// TIA Portal project "010-sps_KnightRider_LightSequencer_tia-portal" (V17)

(* hardware
DEVICE "S7-300/ET200M-Station_1"  S7-300 station
   slot 0: "Profilschiene_0"  Rail  6ES7 390-1***0-0AA0
   slot 1: "PS 307 5A_1"  PS 307 5A  6ES7 307-1EA01-0AA0
   slot 2: "PLC_1"  CPU 314C-2 DP  6ES7 314-6CH04-0AB0  V3.3
      slot 0: "MPI-Schnittstelle_1"  MPI
      slot 1: "DP-Schnittstelle_1"  DP
      slot 2: "DI 24/DO 16_1"  DI24/DO16
      slot 3: "AI 5/AO 2_1"  AI5/AO2
      slot 4: "Zählen_1"  Counter
      slot 5: "Positionieren_1"  Positioning
   slot 4: "DI 16/DO 16x24VDC/0.5A_1"  DI16/DO16 x 24V / 0.5A  6ES7 323-1BL00-0AA0
   slot 5: "DI 16x24VDC_1"  DI16 x 24VDC  6ES7 321-1BH02-0AA0
   slot 6: "CP 342-5_1"  CP 342-5  6GK7 342-5DA03-0XE0  V6.0
   slot 7: "CP 343-1_1"  CP 343-1  6GK7 343-1EX30-0XE0  V2.0
*)

// ===== PLC "PLC_1"  CPU 314C-2 DP =====

VAR_GLOBAL   // PLC tag table "Standard-Variablentabelle"
   "Tag_3" AT %M255.1 : Bool;
   "Start" AT %E0.0 : Bool;
   "Tag_4" AT %M0.0 : Bool;
   "Tag_5" AT %MD10 : DWord;
   "Tag_6" AT %M20.0 : Bool;
   "Tag_7" AT %M0.1 : Bool;
   "Tag_8" AT %M0.2 : Bool;
   "Tag_1" AT %MD30 : DWord;
   "Ausgang" AT %AW0 : Word;
   "Tag_2" AT %AW2 : Word;
   "Tag_9" AT %M255.5 : Bool;
   "Tag_10" AT %M255.3 : Bool;
   "Tag_11" AT %A0.0 : Bool;
   "Tag_12" AT %A124.0 : Bool;
   "Tag_13" AT %A125.0 : Bool;
   "Tag_14" AT %A0.1 : Bool;
END_VAR

DATA_BLOCK "idb10 – Rotieren nach rechts"   // DB10
{ S7_Optimized_Access := 'FALSE' }
VERSION : 0.1
// stored: InstanceOfName FB10 – Rotieren nach rechts-links
"FB10 – Rotieren nach rechts-links"
BEGIN
END_DATA_BLOCK

DATA_BLOCK "idb13 – Lauflichtsteuerung"   // DB13
{ S7_Optimized_Access := 'FALSE' }
VERSION : 0.1
// stored: InstanceOfName FB13 – Lauflichtsteuerung
"FB13 – Lauflichtsteuerung"
BEGIN
END_DATA_BLOCK

DATA_BLOCK "idb15 Night Rider"   // DB15
{ S7_Optimized_Access := 'FALSE' }
VERSION : 0.1
// stored: InstanceOfName FB15 Night Rider
"FB15 Night Rider"
BEGIN
END_DATA_BLOCK

DATA_BLOCK "xdb100 VAR"   // DB100
{ S7_Optimized_Access := 'FALSE' }
VERSION : 0.1
   VAR
      x_Start : Bool;
      w_Src : Word := 1;
      x_clock : Bool;
      w_dest : Word;
   END_VAR
BEGIN
END_DATA_BLOCK

FUNCTION_BLOCK "FB10 – Rotieren nach rechts-links"   // FB10, FBD
{ S7_Optimized_Access := 'FALSE' }
VERSION : 0.1
   VAR_INPUT
      "xStep Val" : Int := 1;
      xClock : Bool;
      xRotierenRechts : Bool;
   END_VAR
   VAR_IN_OUT
      "dw Out Val" : DWord;
   END_VAR
   VAR
      sPtrig1 : Bool;
      sPtrig2 : Bool;
   END_VAR
   VAR_TEMP   // added for the SCL form of the ladder/FBD networks
      _w1 : Bool;
      _w2 : Bool;
   END_VAR
BEGIN

REGION Network 1
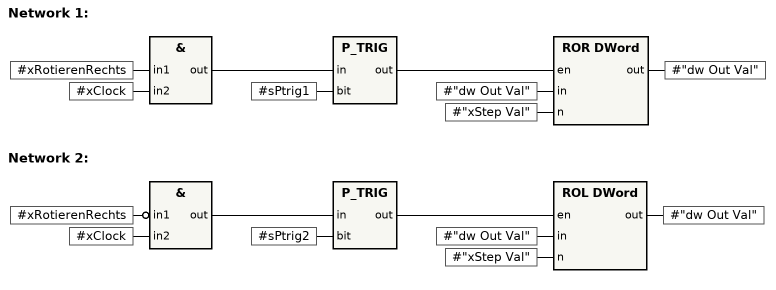
   #_w1 := #xRotierenRechts AND #xClock;
   #_w2 := #_w1 AND NOT #sPtrig1;   // rising edge
   #sPtrig1 := #_w1;
   IF #_w2 THEN #"dw Out Val" := ROR(IN := #"dw Out Val", N := #"xStep Val"); END_IF;
END_REGION

REGION Network 2
   #_w1 := NOT #xRotierenRechts AND #xClock;
   #_w2 := #_w1 AND NOT #sPtrig2;   // rising edge
   #sPtrig2 := #_w1;
   IF #_w2 THEN #"dw Out Val" := ROL(IN := #"dw Out Val", N := #"xStep Val"); END_IF;
END_REGION
END_FUNCTION_BLOCK

FUNCTION_BLOCK "FB13 – Lauflichtsteuerung"   // FB13, FBD
{ S7_Optimized_Access := 'FALSE' }
VERSION : 0.1
   VAR_INPUT
      xStart : Bool;
      xClock : Bool;
   END_VAR
   VAR_OUTPUT
      wAusgänge : Word;
   END_VAR
   VAR_IN_OUT
      "dw Out Val" : DWord;
   END_VAR
   VAR
      xRotateRechts : Bool;
   END_VAR
   VAR_TEMP
      sPtrig : Bool;
      sPtrig_1 : Bool;
      dwRotierterWert : DWord;
   END_VAR
   VAR_TEMP   // added for the SCL form of the ladder/FBD networks
      _w1 : Bool;
   END_VAR
BEGIN

REGION Network 1
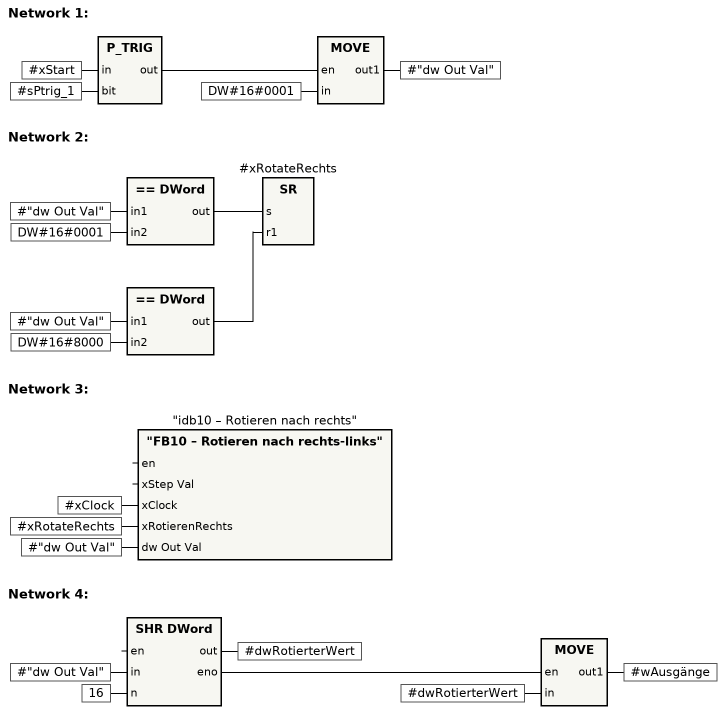
   #_w1 := #xStart AND NOT #sPtrig_1;   // rising edge
   #sPtrig_1 := #xStart;
   IF #_w1 THEN #"dw Out Val" := DW#16#0001; END_IF;
END_REGION

REGION Network 2
   IF #"dw Out Val" = DW#16#0001 THEN
       #xRotateRechts := TRUE;   // SR flip-flop
   END_IF;
   IF #"dw Out Val" = DW#16#8000 THEN #xRotateRechts := FALSE; END_IF;
END_REGION

REGION Network 3
   "idb10 – Rotieren nach rechts"(xClock := #xClock,   // "FB10 – Rotieren nach rechts-links"
                           xRotierenRechts := #xRotateRechts,
                           "dw Out Val" := #"dw Out Val");
END_REGION

REGION Network 4
   // ENO of a box is taken as its EN; it also drops when the box reports an error
   #dwRotierterWert := SHR(IN := #"dw Out Val", N := 16);
   #wAusgänge := #dwRotierterWert;
END_REGION
END_FUNCTION_BLOCK

FUNCTION_BLOCK "FB15 Night Rider"   // FB15, FBD
{ S7_Optimized_Access := 'FALSE' }
VERSION : 0.1
   VAR_INPUT
      x_Start : Bool;
      w_Src : Word;
      x_clock : Bool;
   END_VAR
   VAR_OUTPUT
      w_Dest : Word;
   END_VAR
   VAR
      s_Ptrig_SHL : Bool;
      "s_Ptrig2 NW2" : Bool;
      s_Ptrig_SHR : Bool;
      s_Ptrig_CTUD : Bool;
      IEC_Counter_rechts_links_steuerung : CTUD;
      "x_Control L/R" : Bool;
      w_Dummy_CTUD : Int;
   END_VAR
   VAR_TEMP   // added for the SCL form of the ladder/FBD networks
      _w1 : Bool;
      _w2 : Bool;
   END_VAR
BEGIN

REGION Network 1: werteübergabe am anfang
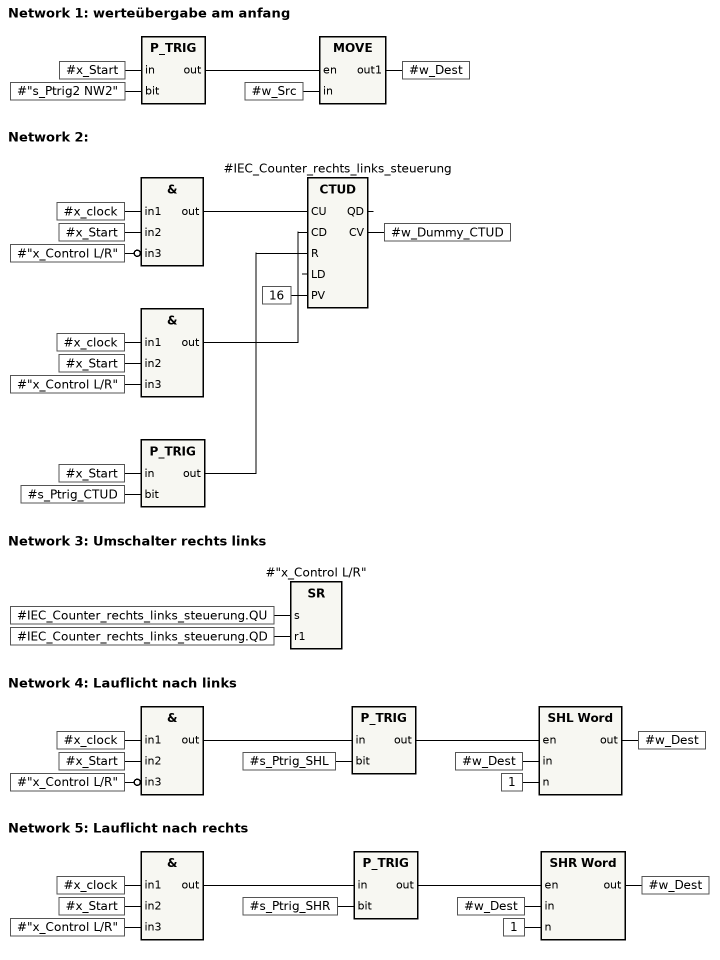
   #_w1 := #x_Start AND NOT #"s_Ptrig2 NW2";   // rising edge
   #"s_Ptrig2 NW2" := #x_Start;
   IF #_w1 THEN #w_Dest := #w_Src; END_IF;
END_REGION

REGION Network 2
   #_w1 := #x_Start AND NOT #s_Ptrig_CTUD;   // rising edge
   #s_Ptrig_CTUD := #x_Start;
   #IEC_Counter_rechts_links_steuerung.CTUD(CU := #x_clock AND #x_Start AND NOT #"x_Control L/R",
                           CD := #x_clock AND #x_Start AND #"x_Control L/R",
                           R := #_w1,
                           PV := 16,
                           CV => #w_Dummy_CTUD);
END_REGION

REGION Network 3: Umschalter rechts links
   IF #IEC_Counter_rechts_links_steuerung.QU THEN
       #"x_Control L/R" := TRUE;   // SR flip-flop
   END_IF;
   IF #IEC_Counter_rechts_links_steuerung.QD THEN #"x_Control L/R" := FALSE; END_IF;
END_REGION

REGION Network 4: Lauflicht nach links
   #_w1 := #x_clock AND #x_Start AND NOT #"x_Control L/R";
   #_w2 := #_w1 AND NOT #s_Ptrig_SHL;   // rising edge
   #s_Ptrig_SHL := #_w1;
   IF #_w2 THEN #w_Dest := SHL(IN := #w_Dest, N := 1); END_IF;
END_REGION

REGION Network 5: Lauflicht nach rechts
   #_w1 := #x_clock AND #x_Start AND #"x_Control L/R";
   #_w2 := #_w1 AND NOT #s_Ptrig_SHR;   // rising edge
   #s_Ptrig_SHR := #_w1;
   IF #_w2 THEN #w_Dest := SHR(IN := #w_Dest, N := 1); END_IF;
END_REGION
END_FUNCTION_BLOCK

ORGANIZATION_BLOCK "Main"   // OB1, FBD
TITLE = "Main Program Sweep (Cycle)"
{ S7_Optimized_Access := 'FALSE' }
VERSION : 0.1
   VAR_TEMP
      OB1_EV_CLASS : Byte;   // Bits 0-3 = 1 (Coming event), Bits 4-7 = 1 (Event class 1)
      OB1_SCAN_1 : Byte;   // 1 (Cold restart scan 1 of OB 1), 3 (Scan 2-n of OB 1)
      OB1_PRIORITY : Byte;   // Priority of OB Execution
      OB1_OB_NUMBR : Byte;   // 1 (Organization block 1, OB1)
      OB1_RESERVED_1 : Byte;   // Reserved for system
      OB1_RESERVED_2 : Byte;   // Reserved for system
      OB1_PREV_CYCLE : Int;   // Cycle time of previous OB1 scan (milliseconds)
      OB1_MIN_CYCLE : Int;   // Minimum cycle time of OB1 (milliseconds)
      OB1_MAX_CYCLE : Int;   // Maximum cycle time of OB1 (milliseconds)
      OB1_DATE_TIME : Date_And_Time;   // Date and time OB1 started
   END_VAR
BEGIN

REGION Network 1
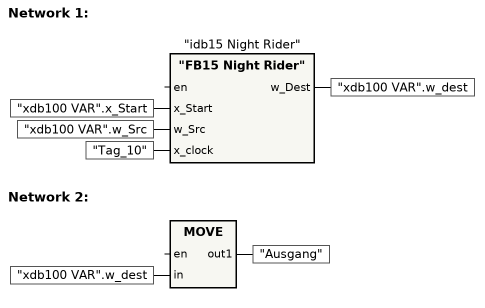
   "idb15 Night Rider"(x_Start := "xdb100 VAR".x_Start,   // "FB15 Night Rider"
                       w_Src := "xdb100 VAR".w_Src,
                       x_clock := "Tag_10",
                       w_Dest => "xdb100 VAR".w_dest);
END_REGION

REGION Network 2
   "Ausgang" := "xdb100 VAR".w_dest;
END_REGION
END_ORGANIZATION_BLOCK